{attribute 'qualified_only'}
VAR_GLOBAL
	//stPlcDriveRef AT %I*: ST_PlcDriveRef;
END_VAR

(* stored: Version 1.1.0.1, ProductVersion 3.1.4022.18
   GVL GVL_IO: Id {f32668ec-d1e3-41ae-be6d-1816d8810958} *)
